SUBAPPLICATION func (* Subapplication Type *)
  (* Standard: 61499-2 *)
  (* Version 1.0, 2025-01-31, franz *)
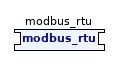
  SUBAPPS
    modbus_rtu : modbus_rtu;
  END_SUBAPPS
END_SUBAPPLICATION
